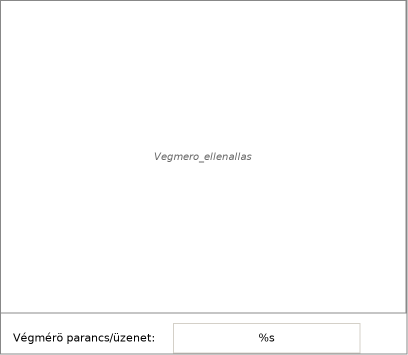
VISUALIZATION Vegmero_auto  // 408x355
    TabControl (0,0 406x313)
        shows Vegmero_ellenallas()
        shows Vegmero_szigeteles()
        shows Vegmero_idoallando()
        shows Vegmero_sokk()
        shows Vegmero_teljes()
        shows Vegmero_etalon()
        [0]: TabTitle=Ellenállás
        [1]: TabTitle=Szigetelés
        [2]: TabTitle=Idöállandó
        [3]: TabTitle=Sokk
        [4]: TabTitle=Teljes/Etalon
        [5]: TabTitle=Etalon
    Textfield (173,323 187x30), "%s", text variable: VEGMERO.s_InCommand
    Label (8,328 150x20), "Végmérö parancs/üzenet:"
END_VISUALIZATION

// ---- VISUs/Vegmero_ellenallas.TcVIS
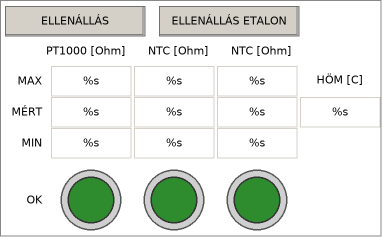
VISUALIZATION Vegmero_ellenallas  // 382x237
    Lamp1 (56,165 70x70), variable: NOT VEGMERO.bPTRES_OK, style: Lamp-Lamp1-Red
    Lamp1 (139,165 70x70), variable: NOT VEGMERO.bNTCRES_OK, style: Lamp-Lamp1-Red
    Button (5,6 140x30), "ELLENÁLLÁS", input disabled if: VEGMERO.s_InCommand<>''
        OnMouseUp: execute { VEGMERO.s_InCommand:='ELLENALLAS'; }
    Textfield (51,97 80x30), "%s", text variable: VEGMERO.rPTRES
    Textfield (134,97 80x30), "%s", text variable: VEGMERO.rNTCRES
    Textfield (51,128 80x30), "%s", text variable: VEGMERO.PTRES_MIN
    Textfield (51,66 80x30), "%s", text variable: VEGMERO.PTRES_MAX
    Textfield (134,128 80x30), "%s", text variable: VEGMERO.NTCRES_MIN
    Textfield (134,66 80x30), "%s", text variable: VEGMERO.NTCRES_MAX
    Textfield (300,97 80x30), "%s", text variable: VEGMERO.rTemp
    Label (5,102 40x20), "MÉRT"
    Label (41,41 90x20), "PT1000 [Ohm]"
    Label (143,41 71x20), "NTC [Ohm]"
    Label (305,70 70x20), "HÖM [C]"
    Button (159,6 140x30), "ELLENÁLLÁS ETALON", input disabled if: VEGMERO.s_InCommand<>''
        OnMouseUp: execute { VEGMERO.s_InCommand:='ELLENALLASETALON'; }
    Label (5,71 40x20), "MAX"
    Label (5,133 40x20), "MIN"
    Label (5,190 40x20), "OK"
    Lamp1 (56,165 70x70), variable: VEGMERO.bPTRES_OK, invisible if: NOT VEGMERO.bPTRES_OK AND VEGMERO.bPTRES_MERVE, style: Lamp-Lamp1-Green
    Lamp1 (139,165 70x70), variable: VEGMERO.bNTCRES_OK, invisible if: NOT VEGMERO.bNTCRES_OK AND VEGMERO.bNTCRES_MERVE, style: Lamp-Lamp1-Green
    Label (226,41 71x20), "NTC [Ohm]"
    Textfield (217,97 80x30), "%s", text variable: VEGMERO.rNTCRES2
    Textfield (217,128 80x30), "%s", text variable: VEGMERO.NTCRES2_MIN
    Textfield (217,66 80x30), "%s", text variable: VEGMERO.NTCRES2_MAX
    Lamp1 (222,165 70x70), variable: NOT VEGMERO.bNTCRES2_OK, style: Lamp-Lamp1-Red
    Lamp1 (222,165 70x70), variable: VEGMERO.bNTCRES2_OK, invisible if: NOT VEGMERO.bNTCRES2_OK AND VEGMERO.bNTCRES2_MERVE, style: Lamp-Lamp1-Green
END_VISUALIZATION

// ---- VISUs/Vegmero_kezi.TcVIS
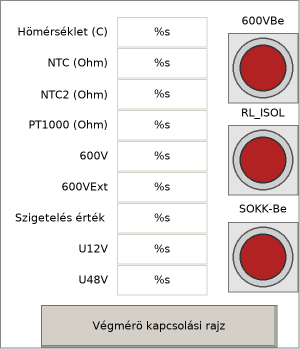
VISUALIZATION Vegmero_kezi  // 300x349
    PushSwitch (228,125 70x70), variable: VEGMERO.bRL_ISOL, behaviour: TOGGLE, style: Switch-PushSwitch-Red
    Label (233,103 60x20), "RL_ISOL"
    Textfield (117,141 90x30), "%s", text variable: VEGMERO.U600V_TRANS
    Textfield (117,48 90x30), "%s", text variable: VEGMERO.NTRES_CALC
    Textfield (117,110 90x30), "%s", text variable: VEGMERO.PTRES_CALC
    Label (11,48 100x30), "NTC (Ohm)"
    Label (11,110 100x30), "PT1000 (Ohm)"
    Label (11,141 100x30), "600V"
    PushSwitch (228,33 70x70), variable: VEGMERO.b600VBe, behaviour: TOGGLE, style: Switch-PushSwitch-Red
    Label (233,11 60x20), "600VBe"
    Textfield (117,265 90x30), "%s", text variable: VEGMERO.U48V_CAL
    Label (11,265 100x30), "U48V"
    Textfield (117,172 90x30), "%s", text variable: VEGMERO.U600VExt_TRANS
    Label (11,172 100x30), "600VExt"
    Textfield (117,203 90x30), "%s", text variable: VEGMERO.UISOL_TRANS
    Label (11,203 97x30), "Szigetelés érték"
    PushSwitch (228,222 70x70), variable: VEGMERO.PT_SOKK48V, behaviour: TOGGLE, style: Switch-PushSwitch-Red
    Label (233,199 60x20), "SOKK-Be"
    Textfield (117,234 90x30), "%s", text variable: VEGMERO.U12V_CAL
    Label (11,234 100x30), "U12V"
    Textfield (117,17 90x30), "%s", text variable: VEGMERO.rHoerzekelo_TRANS
    Label (11,17 100x30), "Hömérséklet (C)"
    Button (41,305 236x42), "Végmérö kapcsolási rajz", tooltip "Ultimate script-ben megírt parancsok pdf-ben", pressed state: Laser.bStartUltimate
        OnMouseUp: execute { VEGMERO.bStartSchematic:=TRUE; }
    Textfield (117,79 90x30), "%s", text variable: VEGMERO.NTRES2_CALC
    Label (11,80 100x30), "NTC2 (Ohm)"
END_VISUALIZATION

// ---- VISUs/Visualization_new.TcVIS
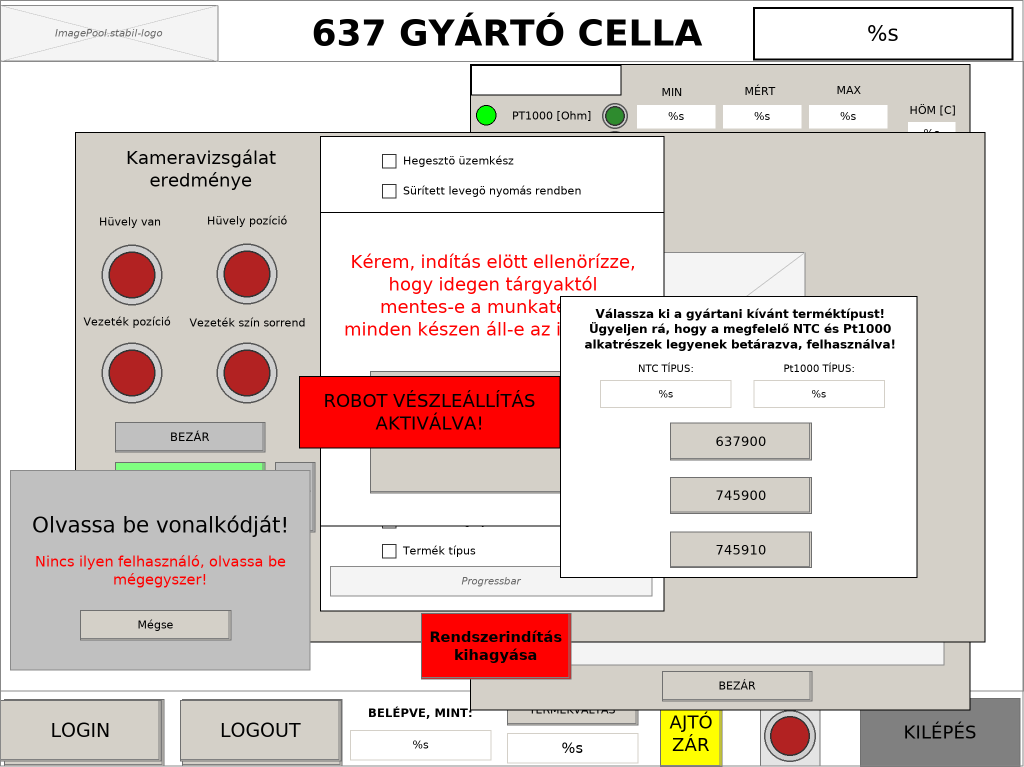
VISUALIZATION Visualization_new  // 1024x767
    Label (518,698 110x30), "TERMÉK TÍPUS:"
    TabControl (0,61 1024x630), invisible if: GVL.bSystemNotStarted, frame switch variable: GVL.iFoLapozo
        shows Termeles0()
        shows Beallitasok()
        shows Szerviz()
        shows TempJozsi()
        shows TempPisti()
        shows Laser()
        shows HegesztesGrafikon()
        [0]: TabTitle=Termelés
        [1]: TabTitle=Beállítások
        [2]: TabTitle=Szervíz
        [3]: TabTitle=Józsi
        [4]: TabTitle=Pisti
        [5]: TabTitle=Lézer
        [6]: TabTitle=Útmérés
    Image (0,5 218x56), image: ImagePool.stabil-logo
    Label (303,9 408x48), "637 GYÁRTÓ CELLA"
    Button (507,695 131x30), "TERMÉKVÁLTÁS"
        OnMouseClick: OpenDialog Dialog=Termektipus, OpenModal=True, OpenCentered=True
    RoundedRectangle (753,7 260x53), "%s", text variable: GVL.sDateTime
    Button (4,699 160x67), "LOGIN", invisible if: true
        OnMouseClick: VisuUserMgmt Type=Login
    Button (860,698 160x69), "KILÉPÉS"
        OnMouseClick: execute { INIT.bStartShutDown:=TRUE; }
    Button (660,700 62x67), "AJTÓ ZÁR", colour toggle: NOT GVL.bBiztonsagiZarBe, pressed state: GVL.bBiztonsagiZarBe, invisible if: NOT INIT.bRobotKesz
        toggle GVL.bBiztonsagiZarGomb
    Textfield (507,733 131x30), "%s", text variable: GVL.sProductType, colour toggle: NOT GVL.bProductTypeOK, input disabled if: true
        OnMouseClick: write the text variable via Edit
    Group (760,690 60x76)
        Label (2,0 55x19), "LEVEGÖ"
        PushSwitch (0,16 60x60), variable: MAIN.bLevego, behaviour: TOGGLE, style: Switch-PushSwitch-Red
    Frame (470,64 500x609), invisible if: GVL.bMeresiEredmenyekRejtve
        shows Meresek()
    Frame (75,132 905x518), invisible if: GVL.bKameraEredmenyekRejtve
        shows Kamera()
    Frame (320,136 149x30), invisible if: GVL.bSystemStarted, input disabled if: GVL.bSystemStarted
        shows Start_ablak()
    Button (182,699 160x67), "LOGOUT", invisible if: true
        OnMouseClick: VisuUserMgmt Type=Logout
    Label (362,698 117x30), "BELÉPVE, MINT:"
    Rectangle (350,730 134x30), "SZERVÍZ"
    Rectangle (350,730 134x30), "FEJLESZTÖ"
    RoundedRectangle (299,376 261x72), "ROBOT VÉSZLEÁLLÍTÁS AKTIVÁLVA!", invisible if: NOT RobotProcess.baStatus[6]
    Textfield (350,730 141x30), "%s", text variable: GVL.UserActual.UserName, input disabled if: true
    Button (0,700 161x61), "LOGIN", input disabled if: GVL.LogButtonsDis
        toggle GVL.LoginEnabled
    Button (180,700 161x61), "LOGOUT", input disabled if: GVL.LogButtonsDis
        toggle GVL.Logout_Button
    Frame (10,470 300x200), invisible if: NOT GVL.LoginEnabled
        shows Login()
END_VISUALIZATION
